// TIA Portal V18 export
FUNCTION "Logica" : Void   // FC1, LAD
{ S7_Optimized_Access := 'TRUE' }
// stored: AutoNumber false, SetENOAutomatically false
   VAR_INPUT
      Richiesta_Lv_1 : Bool;
      Disattiva_Abilitazioni : Bool;
      Password_1 : Array[0..3] of UInt;
   END_VAR
   VAR_OUTPUT
      Livello_1 : Bool;
   END_VAR
   VAR_TEMP   // added for the SCL form of the ladder/FBD networks
      _w1 : Bool;
   END_VAR
BEGIN

REGION Network 1
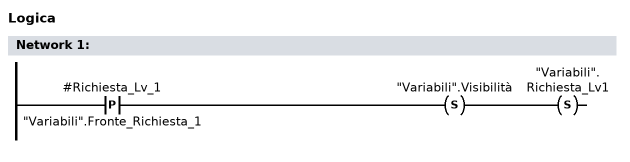
   RUNG wire#powerrail
      P_Contact(operand := #Richiesta_Lv_1, bit := "Variabili".Fronte_Richiesta_1)
      S_Coil( "Variabili".Visibilità )
      S_Coil( "Variabili".Richiesta_Lv1 )
   END_RUNG
   // the same network as SCL:
   #_w1 := #Richiesta_Lv_1 AND NOT "Variabili".Fronte_Richiesta_1;   // rising edge of #Richiesta_Lv_1
   "Variabili".Fronte_Richiesta_1 := #Richiesta_Lv_1;
   IF #_w1 THEN
       "Variabili".Visibilità := TRUE;
       "Variabili".Richiesta_Lv1 := TRUE;
   END_IF;
END_REGION

REGION Network 2 (SCL)
   IF "Variabili".Visibilità = TRUE THEN  //verifico se la visibilità è attiva
       IF "Variabili".Risultato = 0 THEN
             "Variabili".Risultato := 1;
         END_IF;

       IF "Variabili".Conteggio < 4 THEN  //verifico se le volte in cui i numeri sono stati premuti è minore di 4
           //vado a registrare gli input dei pulsanti numerici
           IF ("Variabili".Array_Memoria[0] = true) & ("Variabili".Array_Fronti[0] = false) THEN
                 "Variabili".Array_Input["Variabili".Conteggio] := 0;
                 "Variabili".Conteggio := "Variabili".Conteggio + 1;
             END_IF;

           IF ("Variabili".Array_Memoria[1] = true) & ("Variabili".Array_Fronti[1] = false) THEN
                 "Variabili".Array_Input["Variabili".Conteggio] := 1;
                 "Variabili".Conteggio := "Variabili".Conteggio + 1;
             END_IF;

           IF ("Variabili".Array_Memoria[2] = true) & ("Variabili".Array_Fronti[2] = false) THEN
                 "Variabili".Array_Input["Variabili".Conteggio] := 2;
                 "Variabili".Conteggio := "Variabili".Conteggio + 1;
             END_IF;

           IF ("Variabili".Array_Memoria[3] = true) & ("Variabili".Array_Fronti[3] = false) THEN
                 "Variabili".Array_Input["Variabili".Conteggio] := 3;
                 "Variabili".Conteggio := "Variabili".Conteggio + 1;
             END_IF;

           IF ("Variabili".Array_Memoria[4] = true) & ("Variabili".Array_Fronti[4] = false) THEN
                 "Variabili".Array_Input["Variabili".Conteggio] := 4;
                 "Variabili".Conteggio := "Variabili".Conteggio + 1;
           END_IF;

           IF ("Variabili".Array_Memoria[5] = true) & ("Variabili".Array_Fronti[5] = false) THEN
                 "Variabili".Array_Input["Variabili".Conteggio] := 5;
                 "Variabili".Conteggio := "Variabili".Conteggio + 1;
             END_IF;

           IF ("Variabili".Array_Memoria[6] = true) & ("Variabili".Array_Fronti[6] = false) THEN
                 "Variabili".Array_Input["Variabili".Conteggio] := 6;
                 "Variabili".Conteggio := "Variabili".Conteggio + 1;
             END_IF;

           IF ("Variabili".Array_Memoria[7] = true) & ("Variabili".Array_Fronti[7] = false) THEN
                 "Variabili".Array_Input["Variabili".Conteggio] := 7;
                 "Variabili".Conteggio := "Variabili".Conteggio + 1;
           END_IF;

           IF ("Variabili".Array_Memoria[8] = true) & ("Variabili".Array_Fronti[8] = false) THEN
                 "Variabili".Array_Input["Variabili".Conteggio] := 8;
                 "Variabili".Conteggio := "Variabili".Conteggio + 1;
             END_IF;

           IF ("Variabili".Array_Memoria[9] = true) & ("Variabili".Array_Fronti[9] = false) THEN
                 "Variabili".Array_Input["Variabili".Conteggio] := 9;
                 "Variabili".Conteggio := "Variabili".Conteggio + 1;
           END_IF;

       END_IF;

       IF ("Variabili".Array_Memoria[10] = true) & ("Variabili".Array_Fronti[10] = false) THEN
                   IF "Variabili".Array_Input = #Password_1 THEN
                         "Variabili".Risultato := 2;
                         "Variabili".Livello_1 := true;
                   ELSE
                         "Variabili".Risultato := 3;
                   END_IF;
       END_IF;

       // pressione pulsante "ESC"
       IF ("Variabili".Array_Memoria[11] = true) & ("Variabili".Array_Fronti[11] = false) THEN
            FOR "Variabili".Numero := 0 TO 11 DO
                  "Variabili".Array_Input["Variabili".Numero] := 0;
            END_FOR;
            "Variabili".Conteggio := 0;
            "Variabili".Risultato := 0;
            "Variabili".Visibilità := FALSE;
            "Variabili".Richiesta_Lv1 := false;
       END_IF;

   END_IF;

   IF "Variabili".Livello_1 = true THEN
       #Livello_1 := true;
   END_IF;

   IF #Disattiva_Abilitazioni = true & "Variabili".Fronte_Disabilità = false THEN
       "Variabili".Livello_1 := false;
   END_IF;


   "Variabili".Array_Fronti[0] := "Variabili".Array_Memoria[0];
   "Variabili".Array_Fronti[1] := "Variabili".Array_Memoria[1];
   "Variabili".Array_Fronti[2] := "Variabili".Array_Memoria[2];
   "Variabili".Array_Fronti[3] := "Variabili".Array_Memoria[3];
   "Variabili".Array_Fronti[4] := "Variabili".Array_Memoria[4];
   "Variabili".Array_Fronti[5] := "Variabili".Array_Memoria[5];
   "Variabili".Array_Fronti[6] := "Variabili".Array_Memoria[6];
   "Variabili".Array_Fronti[7] := "Variabili".Array_Memoria[7];
   "Variabili".Array_Fronti[8] := "Variabili".Array_Memoria[8];
   "Variabili".Array_Fronti[9] := "Variabili".Array_Memoria[9];
   "Variabili".Array_Fronti[10] := "Variabili".Array_Memoria[10];
   "Variabili".Array_Fronti[11] := "Variabili".Array_Memoria[11];
   "Variabili".Fronte_Disabilità := #Disattiva_Abilitazioni;
END_REGION
END_FUNCTION
